{attribute 'linkalways'} 
{attribute 'no_explicit_call' := 'This FB is a CLASS and must be accessed using methods or properties'}
{attribute 'enable_dynamic_creation'}
FUNCTION_BLOCK Node_F_VN_ExportSubContainer_String EXTENDS VisionNode
VAR
    ipContainer : _ITcVnContainer;
    nIndex : _ULINT(0);
    sText : _STRING('');
    nMaxLength : _ULINT(0);
    hrPrev : _HRESULT(S_OK);
	hresult : _HRESULT(S_OK);
END_VAR

METHOD PUBLIC  Clone : I_Node
VAR
	pNode : POINTER TO Node_F_VN_ExportSubContainer_String;
END_VAR
pNode := __NEW(Node_F_VN_ExportSubContainer_String);
Clone := pNode^;
END_METHOD

METHOD FB_init : BOOL
VAR_INPUT
	bInitRetains : BOOL; // if TRUE, the retain variables are initialized (warm start / cold start)
	bInCopyCode : BOOL;  // if TRUE, the instance afterwards gets moved into the copy code (online change)
END_VAR
AddInput('ipContainer', ipContainer);
AddParameter('nIndex', nIndex);
AddParameter('nMaxLength', nMaxLength);
AddInput('hrPrev', hrPrev);
AddOutput('sText', sText);
AddOutput('hresult',hresult);
END_METHOD

METHOD PROTECTED OnExecute
hresult.Value := F_VN_ExportSubContainer_String(
	ipContainer := ipContainer.Value,
    nIndex := nIndex.Value,
    sText := sText.Value,
    nMaxLength := nMaxLength.Value,
	hrPrev:= hrPrev.Value);
END_METHOD

METHOD PUBLIC PreExecutionCheck
VAR_INPUT
	Check : I_PreExecutionChecks;
END_VAR
Check.IsTrue(ipContainer.IsValid, 'ipContainer must be a valid container');
Check.IsTrue(ipContainer.IsType(TC_GLOBAL_CONST_LIST.ContainerType_Vector_String_SINT), 'ipContainer contains incorrect type');
END_METHOD

END_FUNCTION_BLOCK

(* stored: Version 1.1.0.1, ProductVersion 3.1.4026.13
   POU Node_F_VN_ExportSubContainer_String: Id {16b442bc-a671-0209-3d46-5bc69b8483fe}, SpecialFunc None
   Folder Constructor: Id {b20c923b-affa-0af9-329d-258aa4afb9b0}
   Method Clone: Id {4b590add-56a7-0e2a-351c-a03be1eacd00}
   Method FB_init: Id {63fdaa99-8371-0ac5-203e-95e469be6259}
   Method OnExecute: Id {f5cf822b-ce7f-0b8b-2e55-2bb899813321}
   Method PreExecutionCheck: Id {529ab91f-4896-0d19-3261-2eff6c988225} *)
